FUNCTION Convert_ULINT_TO_BYTE : Hresult
VAR_INPUT
	in : ULINT;
	out : REFERENCE TO BYTE;
END_VAR
VAR
	converted : BYTE;
END_VAR
VAR CONSTANT
	INCOMPATIBLE : HRESULT := 16#9811070E;
END_VAR

converted := ULINT_TO_BYTE(in);

IF (BYTE_TO_ULINT(converted) <> in) THEN
	Convert_ULINT_TO_BYTE := INCOMPATIBLE;
	RETURN;
END_IF

out := converted;

END_FUNCTION

(* stored: Version 1.1.0.1, ProductVersion 3.1.4024.12
   POU Convert_ULINT_TO_BYTE: Id {9a4a9b07-487c-4e88-b3fe-1c7b39f633db}, SpecialFunc None *)
